{attribute 'linkalways'} 
{attribute 'no_explicit_call' := 'This FB is a CLASS and must be accessed using methods or properties'}
{attribute 'enable_dynamic_creation'}
FUNCTION_BLOCK JsonDeserializerNullForwardEnumerator EXTENDS Disposable IMPLEMENTS I_DeserializerForwardEnumerator, I_EventHandler
VAR
	parent : I_JsonDeserializer;
	nullNode : I_Deserializer;
	invalid : BOOL := FALSE; 
END_VAR

PROPERTY PUBLIC Current : I_Deserializer
GET
Current := nullNode;
END_GET
END_PROPERTY

METHOD FB_exit : BOOL
VAR_INPUT
	bInCopyCode : BOOL; // if TRUE, the exit method is called for exiting an instance that is copied afterwards (online change).
END_VAR
IF bInCopyCode THEN
	RETURN;
END_IF

IF parent = 0 THEN
	RETURN;
END_IF

parent.OffEvent('OnChanged',THIS^);
parent.OffEvent('OnDisposed',THIS^);
END_METHOD

METHOD FB_init : BOOL
VAR_INPUT
	bInitRetains : BOOL; // if TRUE, the retain variables are initialized (warm start / cold start)
	bInCopyCode : BOOL;  // if TRUE, the instance afterwards gets moved into the copy code (online change)
	ParentJsonDeserializer : I_JsonDeserializer;
	ParentNullDeserializer : I_Deserializer;
END_VAR
parent := ParentJsonDeserializer;
nullNode := ParentNullDeserializer;

parent.OnEvent('OnChanged',THIS^);
parent.OnEvent('OnDisposed',THIS^);
END_METHOD

METHOD PUBLIC HandleEvent
VAR_INPUT
	Event : I_Event;
END_VAR
VAR
	changedEvent : I_JsonDeserializerChangedEvent;
	disposedEvent : I_JsonDeserializerDisposedEvent;
END_VAR
IF __QUERYINTERFACE(Event, changedEvent) THEN
	invalid := TRUE;
ELSIF __QUERYINTERFACE(Event, disposedEvent) THEN
	parent := 0;
END_IF
END_METHOD

PROPERTY PUBLIC IsValid : BOOL
GET // PUBLIC
IsValid := (NOT invalid AND parent <> 0);
END_GET
END_PROPERTY

METHOD PUBLIC MoveNext : BOOL
MoveNext := FALSE;
END_METHOD

END_FUNCTION_BLOCK

(* stored: Version 1.1.0.1, ProductVersion 3.1.4024.12
   POU JsonDeserializerNullForwardEnumerator: Id {4b41bc8b-64b2-4cd3-9060-f1d807de7f77}, SpecialFunc None
   Folder Constructor: Id {88b2836c-eeab-4bac-aae5-9a63247a59a6}
   Folder Destructor: Id {5282575f-0f93-4db0-b9d2-b246199d0e1e}
   Property Current: Id {e3529165-dd2e-4849-b130-ef058fb4d0e0}
   Get Get: Id {e7c613a0-aef5-4ab2-b61a-454c5a17cf45}
   Method FB_exit: Id {1728a714-3970-4279-9e23-4955746f5f4f}
   Method FB_init: Id {75ad03d8-a36c-4ab3-83a3-faef44a28444}
   Method HandleEvent: Id {1d9eb21a-9ac6-4ccf-b98d-04e926feb837}
   Property IsValid: Id {b55a7fa5-ccf0-4128-b055-89be113f083e}
   Get Get: Id {74f269be-2365-40f7-acce-b865ef79ad42}
   Method MoveNext: Id {b9dd9ade-fbdf-49f0-996a-e2e8b20500b9} *)
